{attribute 'no_explicit_call' := 'do not call this POU directly'}
FUNCTION_BLOCK INTERNAL FINAL FB_JsonSerializer IMPLEMENTS I_Serializer
VAR_INPUT
END_VAR
VAR_OUTPUT
END_VAR
VAR
	sDataTypeName 	: STRING;
	fbJsonWriter   	: FB_JsonSaxWriter;
	fbJsonDataType 	: FB_JsonReadWriteDataType;
END_VAR

METHOD Serialize : HRESULT
VAR_INPUT
	anyArg	: ANY;
END_VAR
VAR_IN_OUT
	sJsonDocument	: T_VerifyContent;
END_VAR
VAR
	hr : HRESULT;
END_VAR

IF anyArg.diSize <= 0 OR anyArg.pValue = NULL THEN
	// should never happen...
	Serialize := Tc2_System.E_HRESULTAdsErr.INVALIDPARM;
	RETURN;
END_IF

fbJsonWriter.ResetDocument();
sDataTypeName := fbJsonDataType.GetDatatypeNameByAddress(nData:= TO_UDINT(anyArg.diSize), pData:= anyArg.pValue, hrErrorCode=> hr);
IF FAILED(hr) THEN
	Serialize := hr;
	RETURN;
END_IF
fbJsonDataType.AddJsonValueFromSymbol(fbJsonWriter, sDataTypeName , TO_UDINT(anyArg.diSize), anyArg.pValue, hrErrorCode=> hr);
IF FAILED(hr) THEN
	Serialize := hr;
	RETURN;
END_IF
fbJsonWriter.CopyDocument(sJsonDocument, SIZEOF(sJsonDocument) - 1, hrErrorCode=> hr);
IF FAILED(hr) THEN
	Serialize := hr;
	RETURN;
END_IF

IF sJsonDocument = 'null' AND_THEN SUCCEEDED(hr) THEN
	hr := S_FALSE;
END_IF

Serialize := hr;
END_METHOD

END_FUNCTION_BLOCK

(* stored: Version 1.1.0.1, ProductVersion 3.1.4026.18
   POU FB_JsonSerializer: Id {403a942c-72df-482c-961a-a83189084480}, SpecialFunc None
   Method Serialize: Id {1260652b-a648-4fb5-8278-46f89cef46e3} *)
